FUNCTION_BLOCK FINAL FB_TrandChanel
VAR_INPUT 
	UpdatePeriod: TIME:=T#100MS;
	MinimalValue: REAL;
	MaximalValue: REAL:=100;
	TrendType: E_Trend_Visu_Type;
END_VAR
VAR_OUTPUT
	pPoints : POINTER TO ARRAY[0..999] OF VisuStructPoint;
	X_AxisNames : ARRAY [1..10] OF REAL;
	Y_AxisNames : ARRAY [1..15] OF WSTRING(15);
	iPointNumber : INT:=700;
	
END_VAR
VAR_IN_OUT
	TrendChannel: REAL;
END_VAR

VAR
	Timer: TON;
	XY_points : ARRAY[1..1000] OF VisuStructPoint;
	i: INT;
END_VAR

IF UpdatePeriod >= T#100MS THEN
	Timer(IN:=NOT Timer.Q  , PT:= UpdatePeriod);
END_IF

IF TIMER.Q THEN
	X_AxisNames[1]:= MinimalValue;
	X_AxisNames[7]:= MaximalValue;
	FOR i:=2 TO 6 DO
		X_AxisNames[i]:=MinimalValue + ((MaximalValue - MinimalValue)/6)*(i-1);
	END_FOR
	
	FOR i:=1 TO 15 DO
		Y_AxisNames[i]:=TIME_TO_WSTRING_HMI(INT_TO_WORD(i) * UpdatePeriod * 70);
		Y_AxisNames[i]:=WCONCAT("-",Y_AxisNames[i]);
	END_FOR
	
	FOR i:=1 TO 999 DO
		XY_points[1001-i].iY:=XY_points[1000-i].iY;
	END_FOR
	CASE TrendType OF 
		 0: XY_points[1].iY:=450-REAL_TO_INT(TrendChannel*420/(MaximalValue - MinimalValue ));
		 1: 
		(*	xyPoints[1].iY:=210 - REAL_TO_INT(Variable1)*180/100;*)
	END_CASE

END_IF

METHOD FB_init : BOOL
VAR_INPUT
	bInitRetains : BOOL; // if TRUE, the retain variables are initialized (warm start / cold start)
	bInCopyCode : BOOL;  // if TRUE, the instance afterwards gets moved into the copy code (online change)
END_VAR
pPoints:=ADR(XY_points);

FOR i:=1 TO 1000 DO
	XY_points[i].iX:=69+i;
END_FOR
END_METHOD

END_FUNCTION_BLOCK

(* stored: Version 1.1.0.1, ProductVersion 3.1.4024.2
   POU FB_TrandChanel: Id {b3200ce0-00f1-4afb-b8b9-80f3227ead07}, SpecialFunc None
   Method FB_init: Id {1c539689-3422-4e85-aced-5c92c789fc7e} *)
